Universal Robots URScript: gravityFeederV.script

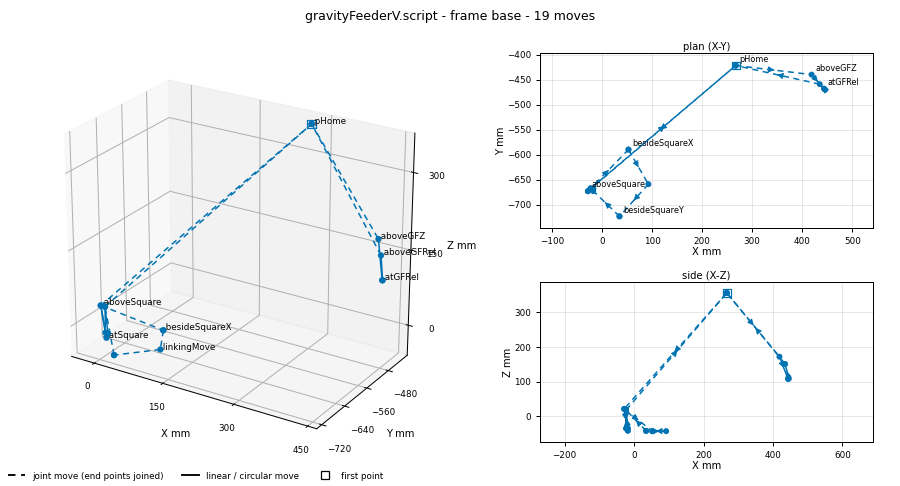
[picture p0: tool path of gravityFeederV.script in frame base, 19 of 21 moves have a stored position in this frame; points joined in program order, loops and branches not executed]
def gravityFeederV():
  set_gravity([0.0, 0.0, 9.82])
  set_tcp(p[0.0,0.0,0.076,0.7245313926163333,-1.7654607319513724,1.7638170400690123])
  set_payload(1.0)
  step_count_7255f790_e5c2_467f_85cd_3e9cf15fcca6 = 0.0
  thread Step_Counter_Thread_663b2e4f_e19b_465f_9f6b_c38d1401a853():
    while (True):
      step_count_7255f790_e5c2_467f_85cd_3e9cf15fcca6 = step_count_7255f790_e5c2_467f_85cd_3e9cf15fcca6 + 1.0
      sync()
    end
  end
  run Step_Counter_Thread_663b2e4f_e19b_465f_9f6b_c38d1401a853()
  set_standard_analog_input_domain(0, 0)
  set_standard_analog_input_domain(1, 0)
  set_tool_analog_input_domain(0, 1)
  set_tool_analog_input_domain(1, 1)
  set_analog_outputdomain(0, 0)
  set_analog_outputdomain(1, 0)
  set_input_actions_to_default()
  set_tool_voltage(0)
  modbus_add_signal("127.0.0.1", 255, 1, 3, "MODBUS_1", False)
  modbus_set_signal_update_frequency("MODBUS_1", 10)
  modbus_add_signal("127.0.0.1", 255, 203, 3, "MODBUS_2", False)
  modbus_set_signal_update_frequency("MODBUS_2", 10)
  modbus_set_runstate_dependent_choice("MODBUS_1",0)
  modbus_set_runstate_dependent_choice("MODBUS_2",0)
  set_safety_mode_transition_hardness(0)
  global stock_spacing=76.2
  global Gravity_Feeder=p[0.26545424739685874,-0.423573422243878,0.3571526050789449,0.1619581347920129,-0.4133494768613531,-2.317499916011395]
  global Linear_Slide=p[0.26542544581166166,-0.4235747955277341,0.35716918848305357,-0.010251867852105759,-0.0039919442596599315,-2.348075206071431]
  # begin: URCap Installation Node
  #   Source: VersaBuilt Robot2CNC, 2.0.9, VersaBuilt Robotics Inc.
  #   Type: R2C Config
  global vbSaveR2CIPAddr = "10.241.34.40"
  global vbSaveDoor = "SingleDoor"
  global vbSaveDoorSensors = True
  global vbSaveDoorWaitTime = 0
  global vbSaveViseSensors = True
  # end: URCap Installation Node
  def _adminLinearIndex2():
    $ 49 "_adminLinearIndex2" "noBreak"
    $ 50 "Move_linear_slide_Index2"
    $ 51 "var_1≔ False "
    global var_1=  False
    $ 52 "Loop var_1≟ False "
    while (var_1 ==   False  ):
      $ 53 "var_1≔socket_open('10.241.34.52',4001)"
      global var_1=socket_open("10.241.34.52",4001)
    end
    $ 54 "var_3≔1"
    global var_3=1
    $ 55 "Send≔'s r0x24 21'"
    global Send="s r0x24 21"
    $ 56 "socket_send_string(Send)"
    socket_send_string(Send)
    $ 57 "socket_send_byte(13)"
    socket_send_byte(13)
    $ 58 "Send_Reply≔socket_read_string()"
    global Send_Reply=socket_read_string()
    $ 59 "Send≔'s r0xca 56389'"
    global Send="s r0xca 56389"
    $ 60 "socket_send_string(Send)"
    socket_send_string(Send)
    $ 61 "socket_send_byte(13)"
    socket_send_byte(13)
    $ 62 "Send_Reply≔socket_read_string()"
    global Send_Reply=socket_read_string()
    $ 63 "Send≔'t 1'"
    global Send="t 1"
    $ 64 "socket_send_string(Send)"
    socket_send_string(Send)
    $ 65 "socket_send_byte(13)"
    socket_send_byte(13)
    $ 66 "Send_Reply≔socket_read_string()"
    global Send_Reply=socket_read_string()
    $ 67 "Loop var_3≠0"
    while (var_3 != 0):
      $ 68 "Send≔'g r0xA0'"
      global Send="g r0xA0"
      $ 69 "socket_send_string(Send)"
      socket_send_string(Send)
      $ 70 "socket_send_byte(13)"
      socket_send_byte(13)
      $ 71 "var_3≔socket_get_var('v')"
      global var_3=socket_get_var("v")
      $ 72 "Wait: 0.1"
      sleep(0.1)
    end
    $ 73 "socket_close()"
    socket_close()
    $ 74 "sync()"
    sync()
  end
  $ 1 "Robot Program"
  $ 2 "Set DO[0]=Off"
  set_standard_digital_out(0, False)
  $ 3 "Call _adminLinearIndex2"
  _adminLinearIndex2()
  $ 4 "MoveJ"
  $ 5 "pHome" "breakAfter"
  movej(get_inverse_kin(p[.267117735476, -.421456669667, .355822513573, 1.114007010937, 1.106163875164, .005128634644], qnear=[-0.7853706518756312, -1.5708320776568812, -1.5708192030536097, -1.5708802382098597, 1.5708121061325073, 4.75623928650748E-5]), a=1.7453292519943295, v=3.141592653589793)
  $ 6 "aboveGFZ" "breakAfter"
  movej(get_inverse_kin(p[.418864874236, -.439594794413, .172117373627, .875334116447, .857585971750, -.012604190968], qnear=[-0.6107004324542444, -1.8580358664142054, -1.839452091847555, -0.6770947615252894, 1.5025687217712402, 0.18094120919704437]), a=1.7453292519943295, v=3.141592653589793)
  $ 7 "MoveL"
  $ 8 "atGFRel" "breakAfter"
  movel(p[.443443169857, -.467485862914, .107996089045, .875451906157, .857812560589, -.012421560532], a=0.05, v=0.15)
  $ 9 "Set DO[0]=On"
  set_standard_digital_out(0, True)
  $ 10 "Wait: 1.0"
  sleep(1.0)
  $ 11 "moveUpRel" "breakAfter"
  movel(p[.445779550876, -.469810205003, .109207315686, .875367578109, .857833002397, -.012511054083], a=0.05, v=0.15)
  $ 12 "aboveGFRel" "breakAfter"
  movel(p[.435113760687, -.458758882872, .151215859232, .875509880483, .857948406618, -.012473289720], a=0.05, v=0.15)
  $ 13 "MoveJ"
  $ 14 "pHome" "breakAfter"
  movej(get_inverse_kin(p[.267117735476, -.421456669667, .355822513573, 1.114007010937, 1.106163875164, .005128634644], qnear=[-0.7853706518756312, -1.5708320776568812, -1.5708192030536097, -1.5708802382098597, 1.5708121061325073, 4.75623928650748E-5]), a=1.7453292519943295, v=3.141592653589793, r=0.1)
  $ 15 "aboveSquare" "breakAfter"
  movej(get_inverse_kin(p[-.028510632568, -.672754849733, .021746809141, 1.706529794651, -.012113432734, -1.206362821846], qnear=[-1.450517479573385, -2.2354820410357874, -1.5772727171527308, -0.8964245955096644, 1.5715678930282593, 0.909832239151001]), a=1.7453292519943295, v=3.141592653589793)
  $ 16 "MoveL"
  $ 17 "atSquare" "breakAfter"
  movel(p[-.017890711485, -.672482386553, -.041426599683, 1.706384217356, -.012380826994, -1.206413833619], a=1.2, v=0.25)
  $ 18 "Set DO[0]=Off"
  set_standard_digital_out(0, False)
  $ 19 "Wait: 0.5"
  sleep(0.5)
  $ 20 "aboveSquare" "breakAfter"
  movel(p[-.028510632568, -.672754849733, .021746809141, 1.706529794651, -.012113432734, -1.206362821846], a=1.2, v=0.25)
  $ 21 "Set DO[0]=On"
  set_standard_digital_out(0, True)
  $ 22 "MoveJ"
  $ 23 "besideSquareX" "breakAfter"
  movej(get_inverse_kin(p[.052617307455, -.589570654624, -.042422525261, 1.706537852760, -.011698760256, -1.207610431296], qnear=[-1.296199146901266, -2.208390537892477, -1.865711514149801, -0.6357458273517054, 1.57034432888031, 1.06466805934906]), a=1.3962634015954636, v=1.0471975511965976)
  $ 24 "MoveL"
  $ 25 "If force()≤40"
  global thread_flag_25=0
  thread Thread_if_25():
    $ 26 "atSquareX" "breakAfter"
    movel(pose_add(get_forward_kin(), pose_sub(p[-.028314437910, -.672474736168, -.041561612947, 1.706659248269, -.012081904034, -1.206394262837], p[.050864659493, -.591008400922, -.041514765275, 1.702232557786, -.007992998753, -1.208859536775])), a=0.035, v=0.035)
    thread_flag_25 = 1
  end
  if ( force () <= 40):
    global thread_handler_25=run Thread_if_25()
    while (thread_flag_25 == 0):
      if not( force () <= 40):
        kill thread_handler_25
        thread_flag_25 = 2
      else:
        sync()
      end
    end
  else:
    thread_flag_25 = 2
  end
  $ 27 "Wait: 0.5"
  sleep(0.5)
  $ 28 "MoveJ"
  $ 29 "besideSquareX" "breakAfter"
  movej(get_inverse_kin(p[.052617307455, -.589570654624, -.042422525261, 1.706537852760, -.011698760256, -1.207610431296], qnear=[-1.296199146901266, -2.208390537892477, -1.865711514149801, -0.6357458273517054, 1.57034432888031, 1.06466805934906]), a=1.3962634015954636, v=1.0471975511965976)
  $ 30 "linkingMove" "breakAfter"
  movej(get_inverse_kin(p[.092406011297, -.658703145464, -.042290441457, 1.707093648604, -.011389994828, -1.206705650649], qnear=[-1.2666195074664515, -2.3227699438678187, -1.6276095549212855, -0.7596004644977015, 1.5709682703018188, 1.0936672687530518]), a=1.3962634015954636, v=1.0471975511965976, r=0.01)
  $ 31 "besideSquareY" "breakAfter"
  movej(get_inverse_kin(p[.034628089998, -.723042022004, -.041529742343, 1.706819891204, -.011779010417, -1.205746278100], qnear=[-1.3717740217791956, -2.423664395009176, -1.416487995778219, -0.8691037336932581, 1.5716880559921265, 0.9880828857421875]), a=1.3962634015954636, v=1.0471975511965976)
  $ 32 "MoveL"
  $ 33 "If force()≤40"
  global thread_flag_33=0
  thread Thread_if_33():
    $ 34 "atSquareY" "breakAfter"
    movel(pose_add(get_forward_kin(), pose_sub(p[-.015805244897, -.673754239162, -.041467023102, 1.706210431136, -.012211069287, -1.206515845875], p[.032384127889, -.724404093144, -.040503922812, 1.702100966605, -.008453431164, -1.209005295943])), a=0.035, v=0.035)
    thread_flag_33 = 1
  end
  if ( force () <= 40):
    global thread_handler_33=run Thread_if_33()
    while (thread_flag_33 == 0):
      if not( force () <= 40):
        kill thread_handler_33
        thread_flag_33 = 2
      else:
        sync()
      end
    end
  else:
    thread_flag_33 = 2
  end
  $ 35 "Wait: 0.5"
  sleep(0.5)
  $ 36 "MoveJ"
  $ 37 "besideSquareY" "breakAfter"
  movej(get_inverse_kin(p[.034628089998, -.723042022004, -.041529742343, 1.706819891204, -.011779010417, -1.205746278100], qnear=[-1.3717740217791956, -2.423664395009176, -1.416487995778219, -0.8691037336932581, 1.5716880559921265, 0.9880828857421875]), a=1.3962634015954636, v=1.0471975511965976)
  $ 38 "aboveSquareNew" "breakAfter"
  movej(get_inverse_kin(p[-.022970780178, -.667274179238, .018449773744, 1.706493853212, -.012107509001, -1.206357709530], qnear=[-1.4411652723895472, -2.229788128529684, -1.5986502806292933, -0.8807080427752894, 1.5715199708938599, 0.9191679954528809]), a=1.3962634015954636, v=1.0471975511965976)
  $ 39 "Set DO[0]=Off"
  set_standard_digital_out(0, False)
  $ 40 "Wait: 1.0"
  sleep(1.0)
  $ 41 "MoveL"
  $ 42 "atSquareNew" "breakAfter"
  movel(p[-.023326599498, -.667602036236, -.034523836862, 1.707778917785, -.043396958913, -1.210750185515], a=1.2, v=0.25)
  $ 43 "Set DO[0]=On"
  set_standard_digital_out(0, True)
  $ 44 "Wait: 1.0"
  sleep(1.0)
  $ 45 "easeout" "breakAfter"
  movel(p[-.017566802315, -.667634704463, -.034572445905, 1.707827808003, -.043421377118, -1.210857271320], a=1.2, v=0.25)
  $ 46 "aboveSquareNew" "breakAfter"
  movel(p[-.022970780178, -.667274179238, .018449773744, 1.706493853212, -.012107509001, -1.206357709530], a=1.2, v=0.25)
  $ 47 "MoveJ"
  $ 48 "pHome" "breakAfter"
  movej(get_inverse_kin(p[.267117735476, -.421456669667, .355822513573, 1.114007010937, 1.106163875164, .005128634644], qnear=[-0.7853706518756312, -1.5708320776568812, -1.5708192030536097, -1.5708802382098597, 1.5708121061325073, 4.75623928650748E-5]), a=1.3962634015954636, v=1.0471975511965976)
end
